ABB RobotStudio station: Task-3.rspag

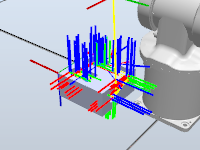
--- station ---
Station Task 3 (saved by RobotStudio 20.1.9056.2)
Controller Controller1
  mechanical unit ROB_1: IRB120_3_58__01, 6 joints, base frame (0, 0, 0) mm
Layout (positions relative to the parent item):
  - IRB120_3_58__01 [mechanism, from Robots\IRB120_3_58_G_01.rslib] at (0, 0, 0) mm; joint values [-0.0516, -0.0762, 0.1853, 0, 1.4617, -1.6224] (rad or m)
  - AssemblyMillCutter_3 [part] at (220.27, 10.34, 568.29) mm, rotated rx -90 ry 0 rz -90 deg
  - Task3_Part [part] at (409.55, -43.91, 250) mm, rotated rx 90 ry 0 rz 90 deg
Attachment: AssemblyMillCutter_3 is attached to IRB120_3_58__01 / Link6
Targets, tools, work objects and paths stored in the station and not in the controller backup, written as RAPID:
! task T_ROB1
MODULE Module1
  CONST robtarget Target_160:=[[-25,64,20],[0,-0.707106781,0.707106781,0],[-1,0,-2,0],[9E+09,9E+09,9E+09,9E+09,9E+09,9E+09]];
  CONST robtarget Target_210:=[[-40,86,20],[0,-0.707106781,0.707106781,0],[-1,0,-2,0],[9E+09,9E+09,9E+09,9E+09,9E+09,9E+09]];
  CONST robtarget Target_220:=[[-40,60,0],[0,0,-0.707106781,0.707106781],[0,0,0,0],[9E+09,9E+09,9E+09,9E+09,9E+09,9E+09]];
  CONST robtarget Target_230:=[[-52.990381057,67.5,0],[0.353553391,-0.353553391,-0.612372436,0.612372436],[0,0,0,0],[9E+09,9E+09,9E+09,9E+09,9E+09,9E+09]];
  CONST robtarget Target_240:=[[-52.990381057,82.5,0],[0.612372436,-0.612372436,-0.353553391,0.353553391],[0,0,0,0],[9E+09,9E+09,9E+09,9E+09,9E+09,9E+09]];
  CONST robtarget Target_250:=[[-40,90,0],[0.707106781,-0.707106781,0,0],[0,0,0,0],[9E+09,9E+09,9E+09,9E+09,9E+09,9E+09]];
ENDMODULE


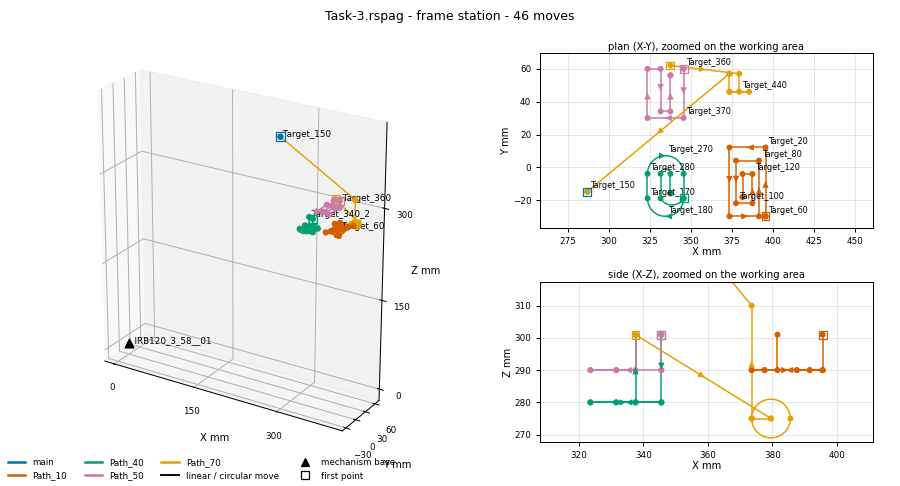
[picture p0: tool path of Task-3.rspag in frame station, 46 of 46 moves have a stored position in this frame; points joined in program order, loops and branches not executed]
--- Backups/Controller1/RAPID/TASK1/PROGMOD/CalibData.mod ---
MODULE CalibData
    TASK PERS tooldata Tooldata_1:=[TRUE,[[-0.002,-0.003,108.338],[0,-0.707106781,0.707106781,0]],[1,[0,0,1],[1,0,0,0],0,0,0]];
    TASK PERS wobjdata Workobject_1:=[FALSE,TRUE,"",[[409.55,-43.91,300],[0,-0.707106781,0.707106781,0]],[[0,0,0],[1,0,0,0]]];
ENDMODULE

--- Backups/Controller1/RAPID/TASK1/PROGMOD/Module1.mod ---
MODULE Module1
        CONST robtarget Target_150:=[[-29.091,122.649,-115.575],[0,-0.707106781,0.707106781,0],[-1,0,-2,0],[9E+09,9E+09,9E+09,9E+09,9E+09,9E+09]];
    CONST robtarget Target_60:=[[-14,14,-1],[0,-0.707106781,0.707106781,0],[-1,0,-2,0],[9E+09,9E+09,9E+09,9E+09,9E+09,9E+09]];
    CONST robtarget Target_10:=[[-14,14,10],[0,-0.707106781,0.707106781,0],[-1,0,-2,0],[9E+09,9E+09,9E+09,9E+09,9E+09,9E+09]];
    CONST robtarget Target_20:=[[-56,14,10],[0,-0.707106781,0.707106781,0],[0,0,-1,0],[9E+09,9E+09,9E+09,9E+09,9E+09,9E+09]];
    CONST robtarget Target_30:=[[-56,36,10],[0,-0.707106781,0.707106781,0],[0,0,-1,0],[9E+09,9E+09,9E+09,9E+09,9E+09,9E+09]];
    CONST robtarget Target_50:=[[-14,36,10],[0,-0.707106781,0.707106781,0],[-1,0,-2,0],[9E+09,9E+09,9E+09,9E+09,9E+09,9E+09]];
    CONST robtarget Target_70:=[[-14,18,10],[0,-0.707106781,0.707106781,0],[-1,0,-2,0],[9E+09,9E+09,9E+09,9E+09,9E+09,9E+09]];
    CONST robtarget Target_80:=[[-48,18,10],[0,-0.707106781,0.707106781,0],[0,0,-1,0],[9E+09,9E+09,9E+09,9E+09,9E+09,9E+09]];
    CONST robtarget Target_90:=[[-48,32,10],[0,-0.707106781,0.707106781,0],[0,0,-1,0],[9E+09,9E+09,9E+09,9E+09,9E+09,9E+09]];
    CONST robtarget Target_100:=[[-22,32,10],[0,-0.707106781,0.707106781,0],[-1,0,-2,0],[9E+09,9E+09,9E+09,9E+09,9E+09,9E+09]];
    CONST robtarget Target_110:=[[-22,22,10],[0,-0.707106781,0.707106781,0],[-1,0,-2,0],[9E+09,9E+09,9E+09,9E+09,9E+09,9E+09]];
    CONST robtarget Target_120:=[[-39.82,22,10],[0,-0.707106781,0.707106781,0],[-1,0,-2,0],[9E+09,9E+09,9E+09,9E+09,9E+09,9E+09]];
    CONST robtarget Target_130:=[[-39.82,28,10],[0,-0.707106781,0.707106781,0],[-1,0,-2,0],[9E+09,9E+09,9E+09,9E+09,9E+09,9E+09]];
    CONST robtarget Target_140:=[[-25.82,28,10],[0,-0.707106781,0.707106781,0],[-1,0,-2,0],[9E+09,9E+09,9E+09,9E+09,9E+09,9E+09]];
    CONST robtarget Target_140_2:=[[-25.82,28,-1],[0,-0.707106781,0.707106781,0],[-1,0,-2,0],[9E+09,9E+09,9E+09,9E+09,9E+09,9E+09]];
    CONST robtarget Target_200:=[[-25,64,-1],[0,-0.707106781,0.707106781,0],[-1,0,-2,0],[9E+09,9E+09,9E+09,9E+09,9E+09,9E+09]];
    CONST robtarget Target_190:=[[-25,64,20],[0,-0.707106781,0.707106781,0],[-1,0,-2,0],[9E+09,9E+09,9E+09,9E+09,9E+09,9E+09]];
    CONST robtarget Target_180:=[[-14,75,20],[0,-0.707106781,0.707106781,0],[-1,0,-2,0],[9E+09,9E+09,9E+09,9E+09,9E+09,9E+09]];
    CONST robtarget Target_170:=[[-25,86,20],[0,-0.707106781,0.707106781,0],[-1,0,-2,0],[9E+09,9E+09,9E+09,9E+09,9E+09,9E+09]];
    CONST robtarget Target_280:=[[-40,86,20],[0,-0.707106781,0.707106781,0],[-1,0,-2,0],[9E+09,9E+09,9E+09,9E+09,9E+09,9E+09]];
    CONST robtarget Target_270:=[[-51,75,20],[0,-0.707106781,0.707106781,0],[0,0,-1,0],[9E+09,9E+09,9E+09,9E+09,9E+09,9E+09]];
    CONST robtarget Target_260:=[[-40,64,20],[0,-0.707106781,0.707106781,0],[-1,0,-2,0],[9E+09,9E+09,9E+09,9E+09,9E+09,9E+09]];
    CONST robtarget Target_290:=[[-22,75,20],[0,-0.707106781,0.707106781,0],[-1,0,-2,0],[9E+09,9E+09,9E+09,9E+09,9E+09,9E+09]];
    CONST robtarget Target_300:=[[-25,78,20],[0,-0.707106781,0.707106781,0],[-1,0,-2,0],[9E+09,9E+09,9E+09,9E+09,9E+09,9E+09]];
    CONST robtarget Target_330:=[[-40,78,20],[0,-0.707106781,0.707106781,0],[-1,0,-2,0],[9E+09,9E+09,9E+09,9E+09,9E+09,9E+09]];
    CONST robtarget Target_310:=[[-43,75,20],[0,-0.707106781,0.707106781,0],[0,0,-1,0],[9E+09,9E+09,9E+09,9E+09,9E+09,9E+09]];
    CONST robtarget Target_320:=[[-40,72,20],[0,-0.707106781,0.707106781,0],[-1,0,-2,0],[9E+09,9E+09,9E+09,9E+09,9E+09,9E+09]];
    CONST robtarget Target_340:=[[-28,72,20],[0,-0.707106781,0.707106781,0],[-1,0,-2,0],[9E+09,9E+09,9E+09,9E+09,9E+09,9E+09]];
    CONST robtarget Target_340_2:=[[-28,72,-1],[0,-0.707106781,0.707106781,0],[-1,0,-2,0],[9E+09,9E+09,9E+09,9E+09,9E+09,9E+09]];
    CONST robtarget Target_360:=[[-104,64,-1],[0,-0.707106781,0.707106781,0],[0,0,-1,0],[9E+09,9E+09,9E+09,9E+09,9E+09,9E+09]];
    CONST robtarget Target_350:=[[-104,64,10],[0,-0.707106781,0.707106781,0],[0,0,0,0],[9E+09,9E+09,9E+09,9E+09,9E+09,9E+09]];
    CONST robtarget Target_370:=[[-74,64,10],[0,-0.707106781,0.707106781,0],[0,0,-1,0],[9E+09,9E+09,9E+09,9E+09,9E+09,9E+09]];
    CONST robtarget Target_380:=[[-74,86,10],[0,-0.707106781,0.707106781,0],[0,0,-1,0],[9E+09,9E+09,9E+09,9E+09,9E+09,9E+09]];
    CONST robtarget Target_390:=[[-104,86,10],[0,-0.707106781,0.707106781,0],[0,0,-1,0],[9E+09,9E+09,9E+09,9E+09,9E+09,9E+09]];
    CONST robtarget Target_400:=[[-104,78,10],[0,-0.707106781,0.707106781,0],[0,0,-1,0],[9E+09,9E+09,9E+09,9E+09,9E+09,9E+09]];
    CONST robtarget Target_410:=[[-78,78,10],[0,-0.707106781,0.707106781,0],[0,0,-1,0],[9E+09,9E+09,9E+09,9E+09,9E+09,9E+09]];
    CONST robtarget Target_420:=[[-78,72,10],[0,-0.707106781,0.707106781,0],[0,0,-1,0],[9E+09,9E+09,9E+09,9E+09,9E+09,9E+09]];
    CONST robtarget Target_430:=[[-100,72,10],[0,-0.707106781,0.707106781,0],[0,0,-1,0],[9E+09,9E+09,9E+09,9E+09,9E+09,9E+09]];
    CONST robtarget Target_430_2:=[[-100,72,-1],[0,-0.707106781,0.707106781,0],[0,0,-1,0],[9E+09,9E+09,9E+09,9E+09,9E+09,9E+09]];
    CONST robtarget Target_430_2_2:=[[-106,72,-1],[0,-0.707106781,0.707106781,0],[0,0,-1,0],[9E+09,9E+09,9E+09,9E+09,9E+09,9E+09]];
    CONST robtarget Target_450:=[[-101,30,25],[0.5,0.5,-0.5,-0.5],[0,0,0,0],[9E+09,9E+09,9E+09,9E+09,9E+09,9E+09]];
    CONST robtarget Target_440:=[[-90,30,25],[0.5,0.5,-0.5,-0.5],[0,-1,-1,0],[9E+09,9E+09,9E+09,9E+09,9E+09,9E+09]];
    CONST robtarget Target_460:=[[-90,36,25],[0.5,0.5,-0.5,-0.5],[0,-1,-1,0],[9E+09,9E+09,9E+09,9E+09,9E+09,9E+09]];
    CONST robtarget Target_470:=[[-90,30,19],[0.5,0.5,-0.5,-0.5],[0,-1,-1,0],[9E+09,9E+09,9E+09,9E+09,9E+09,9E+09]];
    CONST robtarget Target_480:=[[-90,24,25],[0.5,0.5,-0.5,-0.5],[0,-1,-1,0],[9E+09,9E+09,9E+09,9E+09,9E+09,9E+09]];
    CONST robtarget Target_490:=[[-90,30,31],[0.5,0.5,-0.5,-0.5],[0,-1,-1,0],[9E+09,9E+09,9E+09,9E+09,9E+09,9E+09]];
    CONST robtarget Target_500:=[[-90,36,25],[0.5,0.5,-0.5,-0.5],[0,-1,-1,0],[9E+09,9E+09,9E+09,9E+09,9E+09,9E+09]];
    CONST robtarget Target_500_2_2:=[[-101,36,-10],[0.5,0.5,-0.5,-0.5],[0,-1,-1,0],[9E+09,9E+09,9E+09,9E+09,9E+09,9E+09]];
    CONST robtarget Target_500_2:=[[-101,36,25],[0.5,0.5,-0.5,-0.5],[0,-1,-1,0],[9E+09,9E+09,9E+09,9E+09,9E+09,9E+09]];
!***********************************************************
    !
    ! Module:  Module1
    !
    ! Description:
    !   <Insert description here>
    !
    ! Author: miche
    !
    ! Version: 1.0
    !
    !***********************************************************


    !***********************************************************
    !
    ! Procedure main
    !
    !   This is the entry point of your program
    !
    !***********************************************************
    PROC main()
        !Add your code here
        MoveJ Target_150,v20,z0,Tooldata_1\WObj:=Workobject_1;
        Path_10;
    ENDPROC
    PROC Path_10()
        MoveL Target_60,v20,z0,Tooldata_1\WObj:=Workobject_1;
        MoveL Target_10,v20,z0,Tooldata_1\WObj:=Workobject_1;
        MoveL Target_20,v20,z0,Tooldata_1\WObj:=Workobject_1;
        MoveL Target_30,v20,z0,Tooldata_1\WObj:=Workobject_1;
        MoveL Target_50,v20,z0,Tooldata_1\WObj:=Workobject_1;
        MoveL Target_10,v20,z0,Tooldata_1\WObj:=Workobject_1;
        MoveL Target_70,v20,z0,Tooldata_1\WObj:=Workobject_1;
        MoveL Target_80,v20,z0,Tooldata_1\WObj:=Workobject_1;
        MoveL Target_90,v20,z0,Tooldata_1\WObj:=Workobject_1;
        MoveL Target_100,v20,z0,Tooldata_1\WObj:=Workobject_1;
        MoveL Target_110,v20,z0,Tooldata_1\WObj:=Workobject_1;
        MoveL Target_120,v20,z0,Tooldata_1\WObj:=Workobject_1;
        MoveL Target_130,v20,z0,Tooldata_1\WObj:=Workobject_1;
        MoveL Target_140,v20,z0,Tooldata_1\WObj:=Workobject_1;
        MoveL Target_140_2,v20,z0,Tooldata_1\WObj:=Workobject_1;
        Path_40;
    ENDPROC
    PROC Path_40()
        MoveL Target_200,v20,z0,Tooldata_1\WObj:=Workobject_1;
        MoveL Target_190,v20,z0,Tooldata_1\WObj:=Workobject_1;
        MoveC Target_180,Target_170,v20,z0,Tooldata_1\WObj:=Workobject_1;
        MoveL Target_280,v20,z0,Tooldata_1\WObj:=Workobject_1;
        MoveC Target_270,Target_260,v20,z0,Tooldata_1\WObj:=Workobject_1;
        MoveL Target_190,v20,z0,Tooldata_1\WObj:=Workobject_1;
        MoveC Target_290,Target_300,v20,z0,Tooldata_1\WObj:=Workobject_1;
        MoveL Target_330,v20,z0,Tooldata_1\WObj:=Workobject_1;
        MoveC Target_310,Target_320,v20,z0,Tooldata_1\WObj:=Workobject_1;
        MoveL Target_340,v20,z0,Tooldata_1\WObj:=Workobject_1;
        MoveL Target_340_2,v20,z0,Tooldata_1\WObj:=Workobject_1;
        Path_50;
    ENDPROC
    PROC Path_50()
        MoveL Target_360,v20,z0,Tooldata_1\WObj:=Workobject_1;
        MoveL Target_350,v20,z0,Tooldata_1\WObj:=Workobject_1;
        MoveL Target_370,v20,z0,Tooldata_1\WObj:=Workobject_1;
        MoveL Target_380,v20,z0,Tooldata_1\WObj:=Workobject_1;
        MoveL Target_390,v20,z0,Tooldata_1\WObj:=Workobject_1;
        MoveL Target_400,v20,z0,Tooldata_1\WObj:=Workobject_1;
        MoveL Target_410,v20,z0,Tooldata_1\WObj:=Workobject_1;
        MoveL Target_420,v20,z0,Tooldata_1\WObj:=Workobject_1;
        MoveL Target_430,v20,z0,Tooldata_1\WObj:=Workobject_1;
        MoveL Target_430_2,v20,z0,Tooldata_1\WObj:=Workobject_1;
        Path_70;
    ENDPROC
    PROC Path_70()
        MoveL Target_430_2_2,v20,z0,Tooldata_1\WObj:=Workobject_1;
        MoveL Target_450,v20,z0,Tooldata_1\WObj:=Workobject_1;
        MoveL Target_440,v20,z0,Tooldata_1\WObj:=Workobject_1;
        MoveL Target_460,v20,z0,Tooldata_1\WObj:=Workobject_1;
        MoveC Target_470,Target_480,v20,z0,Tooldata_1\WObj:=Workobject_1;
        MoveC Target_490,Target_500,v20,z0,Tooldata_1\WObj:=Workobject_1;
        MoveL Target_500_2,v200,z0,Tooldata_1\WObj:=Workobject_1;
        MoveL Target_500_2_2,v200,z0,Tooldata_1\WObj:=Workobject_1;
        MoveL Target_150,v200,z0,Tooldata_1\WObj:=Workobject_1;
    ENDPROC
ENDMODULE
